FUNCTION_BLOCK XtsEnableSequence IMPLEMENTS ITask
VAR_INPUT
END_VAR
VAR_OUTPUT
END_VAR
VAR
	_collisionGroup : ICollisionGroup;
	addMover : AddMoverToGroupTask(_collisionGroup);
	enableGrp : EnableGroup(_collisionGroup);
	State : INT;
	moverNumbers : DINT;
	AllMoversEnabled: BOOL;
	EnableTrigger : BOOL;
	_busy: BOOL;
	_done: BOOL;
	_Error: BOOL;
END_VAR
VAR_IN_OUT
	arrMovers : ARRAY[*] OF IMover;
END_VAR

CASE State OF
	0:
		IF EnableTrigger THEN
			State := 10;
			EnableTrigger := FALSE;
			moverNumbers := 1;
			_busy := TRUE;
			_done := FALSE;
			_Error := FALSE;
		END_IF
		
	10:
		FOR moverNumbers := LOWER_BOUND(arrMovers,1) TO UPPER_BOUND(arrMovers,1) DO
			arrMovers[moverNumbers].ResetAxis();
		END_FOR
		moverNumbers := 1;
		State := 20;
		
	20:
		IF _collisionGroup.GroupState = CAGroupStatus.mcGroupStateErrorStop THEN
			_collisionGroup.Reset();
		END_IF
		State := 30;
		
	30:
		arrMovers[moverNumbers].IdentInGroup := DINT_TO_INT( moverNumbers);
		IF arrMovers[moverNumbers].AxisRef.NcToPlc.SetPos = 0 THEN
			State := 31;
		END_IF
		addMover.AddMover(MoverToAdd := arrMovers[moverNumbers]);
		State := 40;
		
	40:
		IF addMover.Done THEN
			IF moverNumbers <> UPPER_BOUND(arrMovers,1) THEN
				moverNumbers := moverNumbers + 1;
				State := 30;
			ELSE
				FOR moverNumbers := LOWER_BOUND(arrMovers,1) TO UPPER_BOUND(arrMovers,1) DO
					arrMovers[moverNumbers].EnableAxis();
				END_FOR
				State := 50;
			END_IF
		END_IF
		
	50:
		AllMoversEnabled := TRUE;
		FOR moverNumbers := LOWER_BOUND(arrMovers,1) TO UPPER_BOUND(arrMovers,1) DO
			AllMoversEnabled := TRUE AND arrMovers[moverNumbers].isEnabled();
		END_FOR
		IF AllMoversEnabled THEN
			enableGrp.Execute();
			State := 60;
		END_IF
		
	60:
		IF enableGrp.Done THEN
			State := 0;
			_busy := FALSE;
			_done := true;
		END_IF
END_CASE

addMover();
enableGrp();

METHOD Abort : BOOL
EnableTrigger := FALSE;
State := 0;
addMover.Abort();
enableGrp.Abort();
END_METHOD

PROPERTY Busy : BOOL
GET
Busy := _busy;
END_GET
END_PROPERTY

PROPERTY Done : BOOL
GET
Done := _done;
END_GET
END_PROPERTY

METHOD Enable : BOOL
VAR_INPUT
END_VAR
IF NOT _busy THEN
	EnableTrigger := Enable := true;
END_IF
END_METHOD

PROPERTY Error : BOOL
GET
Error := _Error;
END_GET
END_PROPERTY

METHOD FB_init : BOOL
VAR_INPUT
	bInitRetains : BOOL; // if TRUE, the retain variables are initialized (warm start / cold start)
	bInCopyCode : BOOL;  // if TRUE, the instance afterwards gets moved into the copy code (online change)
	collisionGroup : ICollisionGroup;
END_VAR
_collisionGroup := collisionGroup;
addMover.FB_init(FALSE, FALSE, collisionGroup);
enableGrp.FB_init(FALSE,FALSE, collisionGroup);
END_METHOD

END_FUNCTION_BLOCK

(* stored: Version 1.1.0.1, ProductVersion 3.1.4024.9
   POU XtsEnableSequence: Id {2dbfd422-2e0c-45f9-9282-01bc354cd414}, SpecialFunc None
   Method Abort: Id {d2d6e9f2-aed0-4b3a-a87f-f1996d8a72d7}
   Property Busy: Id {b2847b1e-0ad6-4e6f-aa9c-05b6fa25b442}
   Get Get: Id {cd6105c6-affb-4b98-98f6-bce5ae07cff9}
   Property Done: Id {e08effed-58fa-4696-899c-213c464e3425}
   Get Get: Id {b0ae37c0-67bd-4f74-a37a-4e9cef15bbed}
   Method Enable: Id {f6821b14-22bc-41c2-a356-9ad000e3c73b}
   Property Error: Id {01255016-1bfa-4264-989a-481808856654}
   Get Get: Id {17ab46e5-ad36-493a-89c9-3492f2d2be19}
   Method FB_init: Id {83020818-9cd2-4297-9540-cef3642ab494} *)
